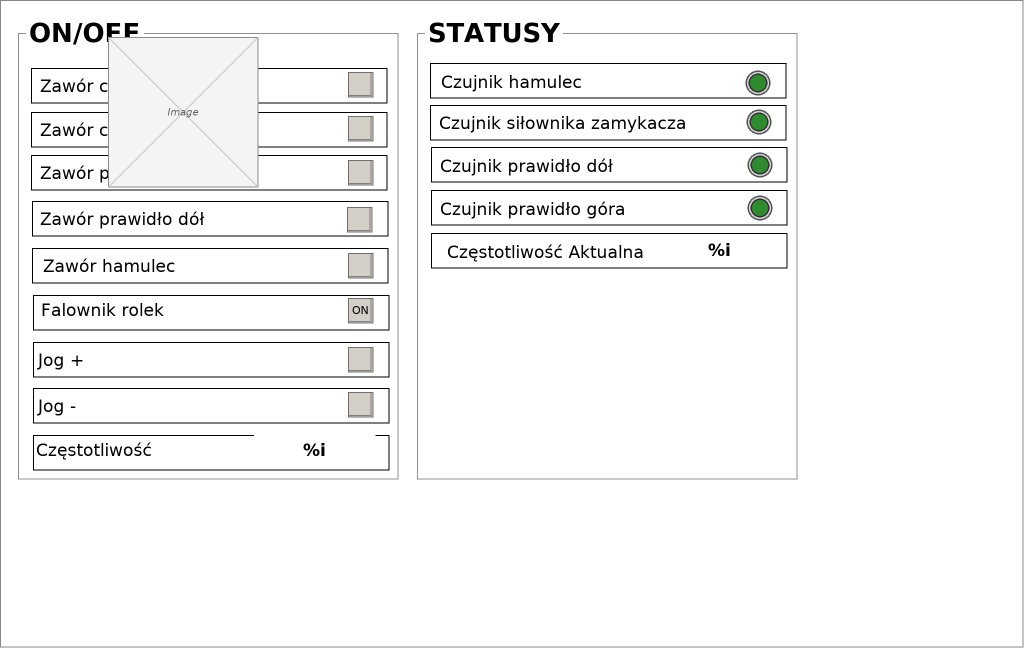
VISUALIZATION Ploter  // 1024x648
    Rectangle (31,155 356x35)
    Label (37,158 208x30), "Zawór prawidło"
    GroupBox (18,25 380x454), "ON/OFF"
        Rectangle (13,43 356x35)
        Rectangle (13,87 356x35)
        Rectangle (15,270 356x35)
        Rectangle (14,223 356x35)
        Label (19,85 239x30)
        Label (19,90 209x30), "Zawór chwytaka 2"
        Label (19,46 209x30), "Zawór chwytaka 1"
        Label (22,226 209x30), "Zawór hamulec"
        Label (20,270 209x30), "Falownik rolek"
        Rectangle (15,410 356x35)
        Label (15,410 216x30), "Częstotliwość"
        Textfield (236,410 121x30), "%i", text variable: GVL_HMI.iWydajnosc
        Button (330,228 25x25), colour toggle: GVL_GLOBAL.zaw_hamulec_cewka
            tap GVL_HMI.przycisk_zaw_hamulec
        Button (330,273 25x25), "ON", colour toggle: GVL_GLOBAL.falownik_rolek_cewka
            tap GVL_HMI.przycisk_falownik_rolek
        Button (330,91 25x25), colour toggle: GVL_GLOBAL.zaw_chwyt2_cewka
            tap GVL_HMI.przycisk_zaw_chwyt2
        Button (330,47 25x25), colour toggle: GVL_GLOBAL.zaw_chwyt1_cewka
            tap GVL_HMI.przycisk_zaw_chwyt1
        Rectangle (14,176 356x35)
        Button (330,135 25x25), colour toggle: GVL_GLOBAL.zaw_prawidlo_cewka
            tap GVL_HMI.przycisk_zaw_prawidlo
        Button (329,182 25x25), colour toggle: GVL_GLOBAL.zaw_prawidlo_dol_cewka
            tap GVL_HMI.przycisk_zaw_prawdidlo_dol
        Rectangle (15,317 356x35)
        Rectangle (15,363 356x35)
        Label (17,320 209x30), "Jog +"
        Label (17,366 209x30), "Jog -"
        Button (330,322 25x25), colour toggle: GVL_GLOBAL.zaw_hamulec_cewka
            tap GVL_HMI.bHmiPlotCCw
        Button (330,367 25x25), colour toggle: GVL_GLOBAL.zaw_hamulec_cewka
            tap GVL_HMI.bHmiPlotCw
    Image (108,37 150x150)
    GroupBox (417,25 380x454), "STATUSY"
        Rectangle (13,38 356x35)
        Label (19,41 230x30)
        Rectangle (13,80 356x35)
        Label (19,83 239x30), "Czujnik siłownika zamykacza"
        Lamp1 (328,83 28x28), variable: GVL_IO_P.b3B1, style: Lamp-Lamp1-Green
        Lamp1 (327,44 28x28), variable: GVL_IO_P.b5B1, style: Lamp-Lamp1-Green
        Label (21,42 239x30), "Czujnik hamulec"
        Rectangle (14,122 356x35)
        Rectangle (14,165 356x35)
        Rectangle (14,208 356x35)
        Label (27,212 209x30), "Częstotliwość Aktualna"
        Textfield (242,210 121x30), "%i", text variable: GVL_HMI.iWydajnosc
    Label (437,151 239x30), "Czujnik prawidło dół"
    Lamp1 (746,151 28x28), variable: GVL_IO_P.b2B1, style: Lamp-Lamp1-Green
    Label (437,194 239x30), "Czujnik prawidło góra"
    Lamp1 (746,194 28x28), variable: GVL_IO_P.b6B1, style: Lamp-Lamp1-Green
    Label (37,204 212x30), "Zawór prawidło dół"
END_VISUALIZATION

(* stored: Version 1.1.0.1, ProductVersion 3.1.4022.12
   Visu Ploter: Id {1286ed3c-bb5c-400d-8c8a-0b3226d12254} *)
